(* Logix 5000 project; controller Project_Template vendor 1 type 14 code 106 rev 33.11; software revision 33.00 *)

TASK MainTask (continuous, watchdog 500 ms) : MainProgram

MODULES
   Local : vendor 1 type 14 code 106 (Compact 0, rev 33.11)
      Discrete_In_Slot_3 : 1769-IQ16 (Compact 3, rev 1.1, Input RPI 20 ms)
      Discrete_In_Slot_2 : 1769-IQ16 (Compact 2, rev 1.1, Input RPI 20 ms)
      Discrete_Out_Slot_5 : 1769-OW16 (Compact 5, rev 1.1, Output RPI 20 ms)
      Discrete_Out_Slot_4 : 1769-OW16 (Compact 4, rev 1.1, Output RPI 20 ms)
      ASCII_Slot_1 : vendor 1 type 109 code 66 (Compact 1, rev 2.1, Output RPI 2 ms)
END_MODULES

TYPE BCR_Data :
STRUCT
   LEN : DINT;
   DATA : SINT[9];
END_STRUCT
END_TYPE

TYPE Color_Data :
STRUCT
   LEN : DINT;
   DATA : SINT[4];
END_STRUCT
END_TYPE

VAR_GLOBAL   (* controller tags *)
   I_Auto_Mode_Selector : ALIAS FOR Local:2:I.Data.2;
   I_Barcode_Stop_Raised : ALIAS FOR Local:3:I.Data.1;
   I_Box_Ejector_Extended : ALIAS FOR Local:2:I.Data.4;
   I_Exit_Proxy : ALIAS FOR Local:3:I.Data.7;
   I_Reject_Cyl_Lowered : ALIAS FOR Local:3:I.Data.2;
   I_Reset_PB : ALIAS FOR Local:2:I.Data.3;
   I_Start_PB : ALIAS FOR Local:2:I.Data.0;
   I_Stop_PB : ALIAS FOR Local:2:I.Data.1;
   I_Vacuum_Head_at_Conveyor : ALIAS FOR Local:3:I.Data.0;
   I_Vacuum_Head_at_Magazine : ALIAS FOR Local:2:I.Data.15;
   I_Vacuum_Head_Extended : ALIAS FOR Local:2:I.Data.14;
   I_Vacuum_Head_Lowered : ALIAS FOR Local:2:I.Data.10;
   I_Vacuum_Head_Raised : ALIAS FOR Local:2:I.Data.9;
   I_Vacuum_Head_Retracted : ALIAS FOR Local:2:I.Data.13;
   I_Vacuum_Head_Rotated_CCW : ALIAS FOR Local:2:I.Data.11;
   I_Vacuum_Head_Rotated_CW : ALIAS FOR Local:2:I.Data.12;
   I_Vacuum_Sensor_On : ALIAS FOR Local:3:I.Data.8;
   O_Amber_Tower_Ind : ALIAS FOR Local:5:O.Data.9;
   O_Barcode_Stop_Raise : ALIAS FOR Local:4:O.Data.14;
   O_Box_Eject : ALIAS FOR Local:4:O.Data.0;
   O_Conveyor_On : ALIAS FOR Local:5:O.Data.5;
   O_Green_Tower_Ind : ALIAS FOR Local:5:O.Data.8;
   O_Red_Tower_Ind : ALIAS FOR Local:5:O.Data.10;
   O_Reject_Cyl_Extend : ALIAS FOR Local:5:O.Data.0;
   O_Reject_Cyl_Lower : ALIAS FOR Local:4:O.Data.15;
   O_Vacuum_Head_Extend : ALIAS FOR Local:4:O.Data.8;
   O_Vacuum_Head_Lower : ALIAS FOR Local:4:O.Data.5;
   O_Vacuum_Head_Rotate_CCW : ALIAS FOR Local:4:O.Data.7;
   O_Vacuum_Head_Rotate_CW : ALIAS FOR Local:4:O.Data.6;
   O_Vacuum_Head_to_Conveyor : ALIAS FOR Local:4:O.Data.9;
   O_Vacuum_Head_to_Magazine : ALIAS FOR Local:4:O.Data.10;
   O_Vacuum_Off : ALIAS FOR Local:5:O.Data.2;
   O_Vacuum_On : ALIAS FOR Local:5:O.Data.1;
END_VAR

PROGRAM MainProgram   (* main routine MainRoutine *)
VAR
   BCR_Good_Read : BOOL;
   BCR_Value : BCR_Data := '33320359$0D';
   Box_Filtered : BOOL;
   Color_Code : DINT := 2;
   Color_Value : Color_Data := '2';
   Delay_Timer : TIMER := (PRE := 3000);
   Fast_Flash_Off : TIMER := (PRE := 250, ACC := 182, EN := 1, TT := 1);
   Fast_Flash_On : TIMER := (PRE := 250, ACC := 250, EN := 1, DN := 1);
   Fast_Flasher : BOOL := 1;
   Filter_Done : BOOL := 1;
   Home_Verify : BOOL;
   Machine_Home : BOOL;
   New_Rx_ID : SINT := 26;
   Normal_Flash_Off : TIMER := (PRE := 500);
   Normal_Flash_On : TIMER := (PRE := 500, ACC := 432, EN := 1, TT := 1);
   Old_Rx_ID : SINT := 26;
   Prod_Cycl_Cntr : COUNTER := (ACC := 4, CU := 1, DN := 1);
   Prod_Cycl_end : BOOL := 1;
   Prod_Running : BOOL;
   Prod_Step : DINT;
   Prod_Test_Bit : DINT := -1;
   Production : BOOL;
   Regular_flasher : BOOL;
   Reject_Box : BOOL;
   Reset_Delay_Timer : TIMER[10] := ([0].PRE := 1000, [1].PRE := 1000, [2].PRE := 1000, [3].PRE := 1000, [4].PRE := 1000, [4].ACC := 1000, [4].EN := 1, [4].DN := 1, [5].PRE := 1000, [5].ACC := 1000, [5].EN := 1, [5].DN := 1);
   Reset_step : DINT;
   Reset_Test_Bit : DINT := -1;
   Resetting : BOOL;
   Rotate_timer : TIMER := (PRE := 500);
   Slow_Flash_Off : TIMER := (PRE := 1000);
   Slow_Flash_ON : TIMER := (PRE := 1000, ACC := 432, EN := 1, TT := 1);
   Slow_Flasher : BOOL;
   Stop_Bit : BOOL;
   Test_Bit : DINT;
END_VAR

ROUTINE a_Reset_Routine   (* ladder *)
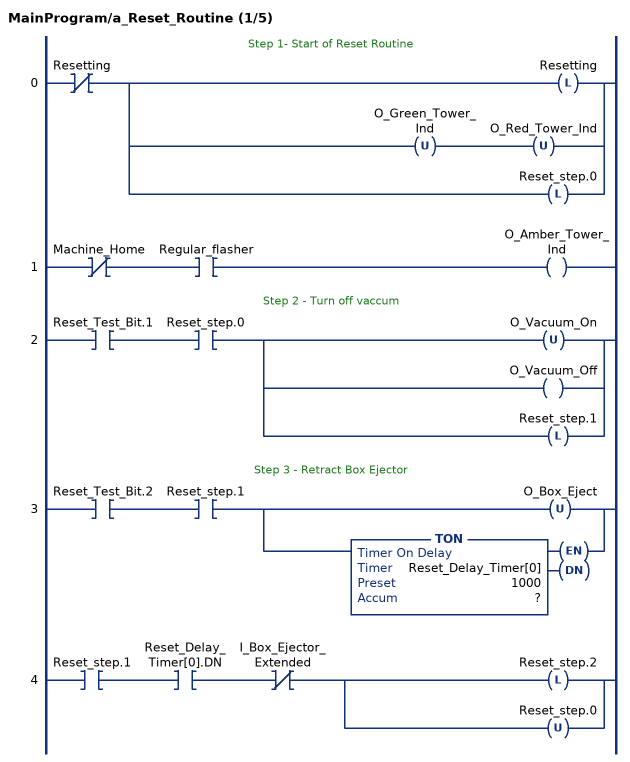
   // Step 1- Start of Reset Routine
   0: XIO(Resetting)[OTL(Resetting) ,OTU(O_Green_Tower_Ind) OTU(O_Red_Tower_Ind) ,OTL(Reset_step.0) ];
   1: XIO(Machine_Home)XIC(Regular_flasher)OTE(O_Amber_Tower_Ind);
   // Step 2 - Turn off vaccum
   2: XIC(Reset_Test_Bit.1)XIC(Reset_step.0)[OTU(O_Vacuum_On) ,OTE(O_Vacuum_Off) ,OTL(Reset_step.1) ];
   // Step 3 - Retract Box Ejector
   3: XIC(Reset_Test_Bit.2)XIC(Reset_step.1)[OTU(O_Box_Eject) ,TON(Reset_Delay_Timer[0],?,?) ];
   4: XIC(Reset_step.1)XIC(Reset_Delay_Timer[0].DN)XIO(I_Box_Ejector_Extended)[OTL(Reset_step.2) ,OTU(Reset_step.0) ];
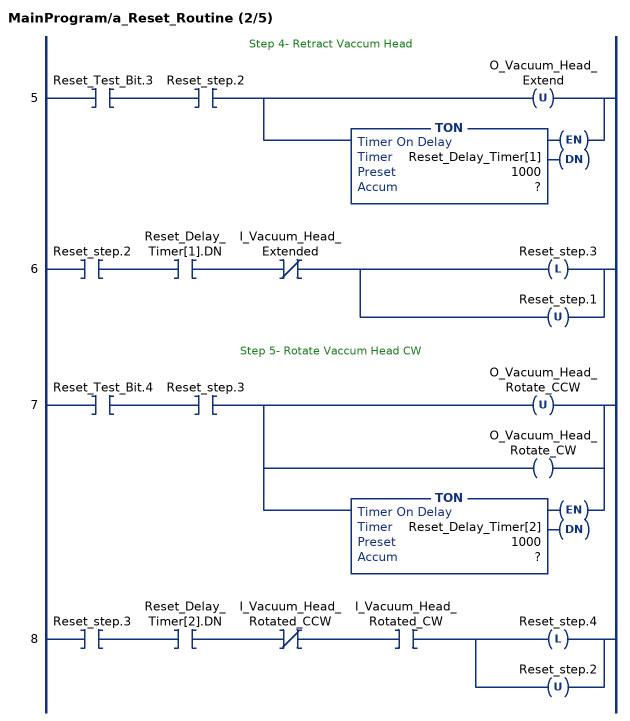
   // Step 4- Retract Vaccum Head
   5: XIC(Reset_Test_Bit.3)XIC(Reset_step.2)[OTU(O_Vacuum_Head_Extend) ,TON(Reset_Delay_Timer[1],?,?) ];
   6: XIC(Reset_step.2)XIC(Reset_Delay_Timer[1].DN)XIO(I_Vacuum_Head_Extended)[OTL(Reset_step.3) ,OTU(Reset_step.1) ];
   // Step 5- Rotate Vaccum Head CW
   7: XIC(Reset_Test_Bit.4)XIC(Reset_step.3)[OTU(O_Vacuum_Head_Rotate_CCW) ,OTE(O_Vacuum_Head_Rotate_CW) ,TON(Reset_Delay_Timer[2],?,?) ];
   8: XIC(Reset_step.3)XIC(Reset_Delay_Timer[2].DN)XIO(I_Vacuum_Head_Rotated_CCW)XIC(I_Vacuum_Head_Rotated_CW)[OTL(Reset_step.4) ,OTU(Reset_step.2) ];
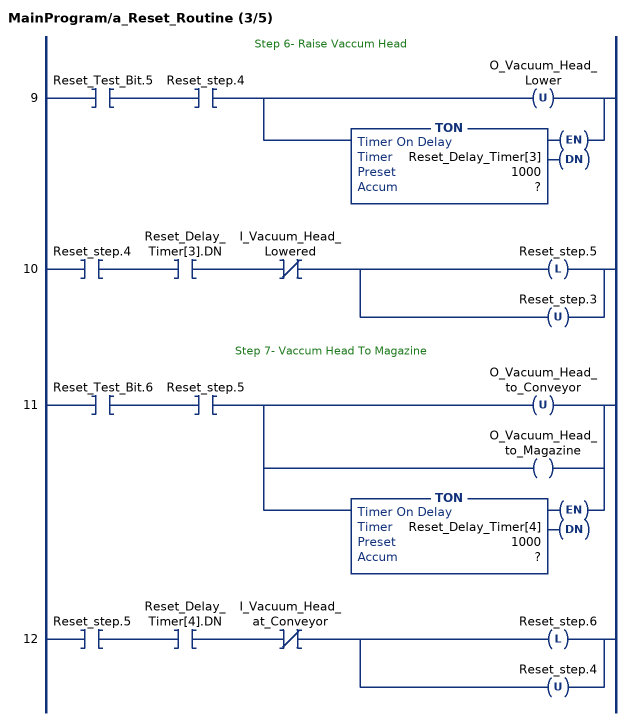
   // Step 6- Raise Vaccum Head
   9: XIC(Reset_Test_Bit.5)XIC(Reset_step.4)[OTU(O_Vacuum_Head_Lower) ,TON(Reset_Delay_Timer[3],?,?) ];
   10: XIC(Reset_step.4)XIC(Reset_Delay_Timer[3].DN)XIO(I_Vacuum_Head_Lowered)[OTL(Reset_step.5) ,OTU(Reset_step.3) ];
   // Step 7- Vaccum Head To Magazine
   11: XIC(Reset_Test_Bit.6)XIC(Reset_step.5)[OTU(O_Vacuum_Head_to_Conveyor) ,OTE(O_Vacuum_Head_to_Magazine) ,TON(Reset_Delay_Timer[4],?,?) ];
   12: XIC(Reset_step.5)XIC(Reset_Delay_Timer[4].DN)XIO(I_Vacuum_Head_at_Conveyor)[OTL(Reset_step.6) ,OTU(Reset_step.4) ];
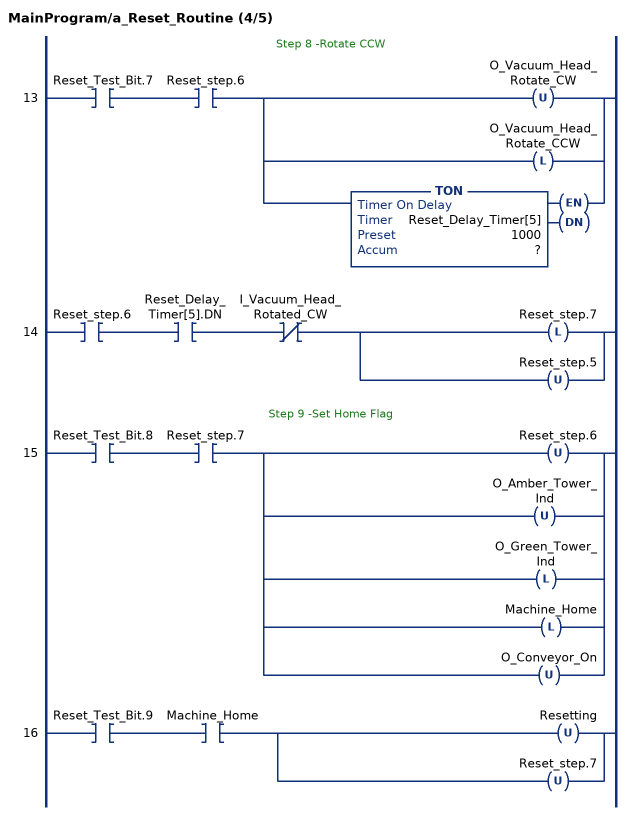
   // Step 8 -Rotate CCW
   13: XIC(Reset_Test_Bit.7)XIC(Reset_step.6)[OTU(O_Vacuum_Head_Rotate_CW) ,OTL(O_Vacuum_Head_Rotate_CCW) ,TON(Reset_Delay_Timer[5],?,?) ];
   14: XIC(Reset_step.6)XIC(Reset_Delay_Timer[5].DN)XIO(I_Vacuum_Head_Rotated_CW)[OTL(Reset_step.7) ,OTU(Reset_step.5) ];
   // Step 9 -Set Home Flag
   15: XIC(Reset_Test_Bit.8)XIC(Reset_step.7)[OTU(Reset_step.6) ,OTU(O_Amber_Tower_Ind) ,OTL(O_Green_Tower_Ind) ,OTL(Machine_Home) ,OTU(O_Conveyor_On) ];
   16: XIC(Reset_Test_Bit.9)XIC(Machine_Home)[OTU(Resetting) ,OTU(Reset_step.7) ];
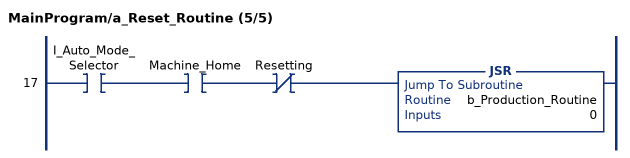
   17: XIC(I_Auto_Mode_Selector)XIC(Machine_Home)XIO(Resetting)JSR(b_Production_Routine,0);
END_ROUTINE

ROUTINE b_Production_Routine   (* ladder *)
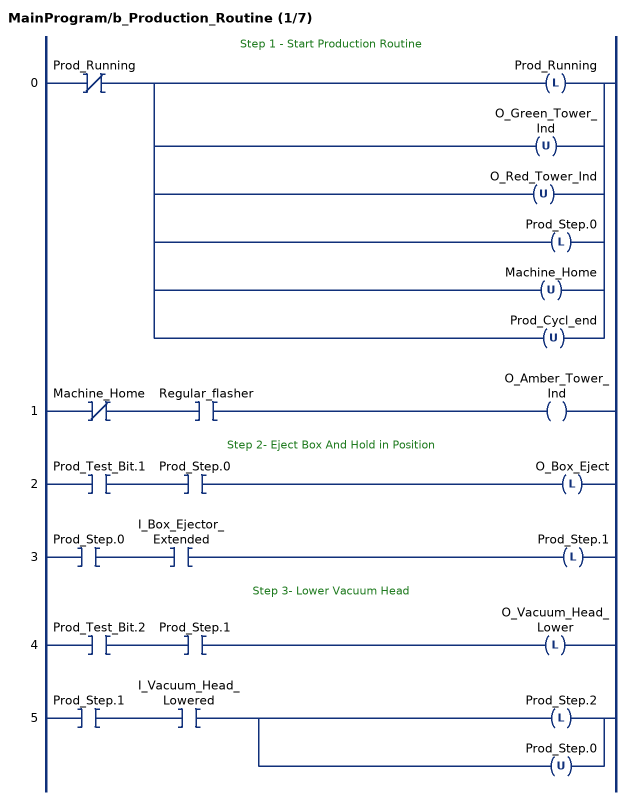
   // Step 1 - Start Production Routine
   0: XIO(Prod_Running)[OTL(Prod_Running) ,OTU(O_Green_Tower_Ind) ,OTU(O_Red_Tower_Ind) ,OTL(Prod_Step.0) ,OTU(Machine_Home) ,OTU(Prod_Cycl_end) ];
   1: XIO(Machine_Home)XIC(Regular_flasher)OTE(O_Amber_Tower_Ind);
   // Step 2- Eject Box And Hold in Position
   2: XIC(Prod_Test_Bit.1)XIC(Prod_Step.0)OTL(O_Box_Eject);
   3: XIC(Prod_Step.0)XIC(I_Box_Ejector_Extended)OTL(Prod_Step.1);
   // Step 3- Lower Vacuum Head
   4: XIC(Prod_Test_Bit.2)XIC(Prod_Step.1)OTL(O_Vacuum_Head_Lower);
   5: XIC(Prod_Step.1)XIC(I_Vacuum_Head_Lowered)[OTL(Prod_Step.2) ,OTU(Prod_Step.0) ];
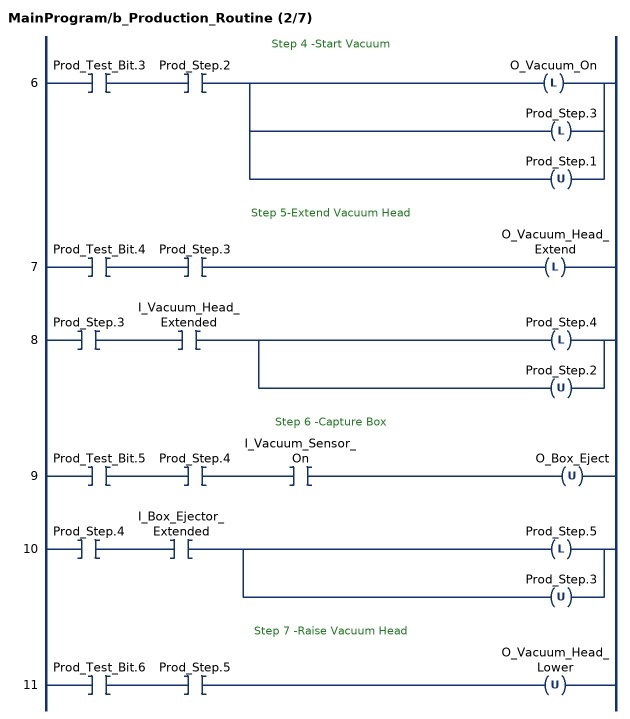
   // Step 4 -Start Vacuum
   6: XIC(Prod_Test_Bit.3)XIC(Prod_Step.2)[OTL(O_Vacuum_On) ,OTL(Prod_Step.3) ,OTU(Prod_Step.1) ];
   // Step 5-Extend Vacuum Head
   7: XIC(Prod_Test_Bit.4)XIC(Prod_Step.3)OTL(O_Vacuum_Head_Extend);
   8: XIC(Prod_Step.3)XIC(I_Vacuum_Head_Extended)[OTL(Prod_Step.4) ,OTU(Prod_Step.2) ];
   // Step 6 -Capture Box
   9: XIC(Prod_Test_Bit.5)XIC(Prod_Step.4)XIC(I_Vacuum_Sensor_On)OTU(O_Box_Eject);
   10: XIC(Prod_Step.4)XIC(I_Box_Ejector_Extended)[OTL(Prod_Step.5) ,OTU(Prod_Step.3) ];
   // Step 7 -Raise Vacuum Head
   11: XIC(Prod_Test_Bit.6)XIC(Prod_Step.5)OTU(O_Vacuum_Head_Lower);
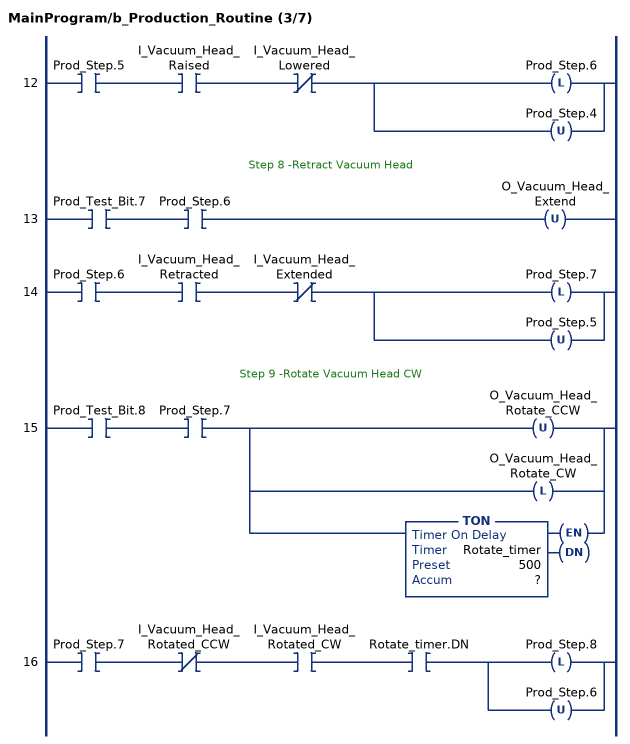
   12: XIC(Prod_Step.5)XIC(I_Vacuum_Head_Raised)XIO(I_Vacuum_Head_Lowered)[OTL(Prod_Step.6) ,OTU(Prod_Step.4) ];
   // Step 8 -Retract Vacuum Head
   13: XIC(Prod_Test_Bit.7)XIC(Prod_Step.6)OTU(O_Vacuum_Head_Extend);
   14: XIC(Prod_Step.6)XIC(I_Vacuum_Head_Retracted)XIO(I_Vacuum_Head_Extended)[OTL(Prod_Step.7) ,OTU(Prod_Step.5) ];
   // Step 9 -Rotate Vacuum Head CW
   15: XIC(Prod_Test_Bit.8)XIC(Prod_Step.7)[OTU(O_Vacuum_Head_Rotate_CCW) ,OTL(O_Vacuum_Head_Rotate_CW) ,TON(Rotate_timer,?,?) ];
   16: XIC(Prod_Step.7)XIO(I_Vacuum_Head_Rotated_CCW)XIC(I_Vacuum_Head_Rotated_CW)XIC(Rotate_timer.DN)[OTL(Prod_Step.8) ,OTU(Prod_Step.6) ];
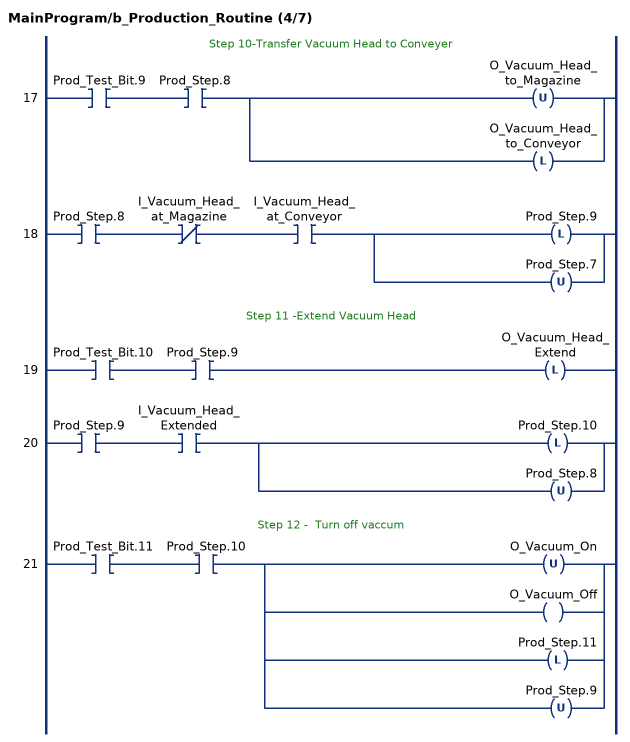
   // Step 10-Transfer Vacuum Head to Conveyer
   17: XIC(Prod_Test_Bit.9)XIC(Prod_Step.8)[OTU(O_Vacuum_Head_to_Magazine) ,OTL(O_Vacuum_Head_to_Conveyor) ];
   18: XIC(Prod_Step.8)XIO(I_Vacuum_Head_at_Magazine)XIC(I_Vacuum_Head_at_Conveyor)[OTL(Prod_Step.9) ,OTU(Prod_Step.7) ];
   // Step 11 -Extend Vacuum Head
   19: XIC(Prod_Test_Bit.10)XIC(Prod_Step.9)OTL(O_Vacuum_Head_Extend);
   20: XIC(Prod_Step.9)XIC(I_Vacuum_Head_Extended)[OTL(Prod_Step.10) ,OTU(Prod_Step.8) ];
   // Step 12 -  Turn off vaccum
   21: XIC(Prod_Test_Bit.11)XIC(Prod_Step.10)[OTU(O_Vacuum_On) ,OTE(O_Vacuum_Off) ,OTL(Prod_Step.11) ,OTU(Prod_Step.9) ];
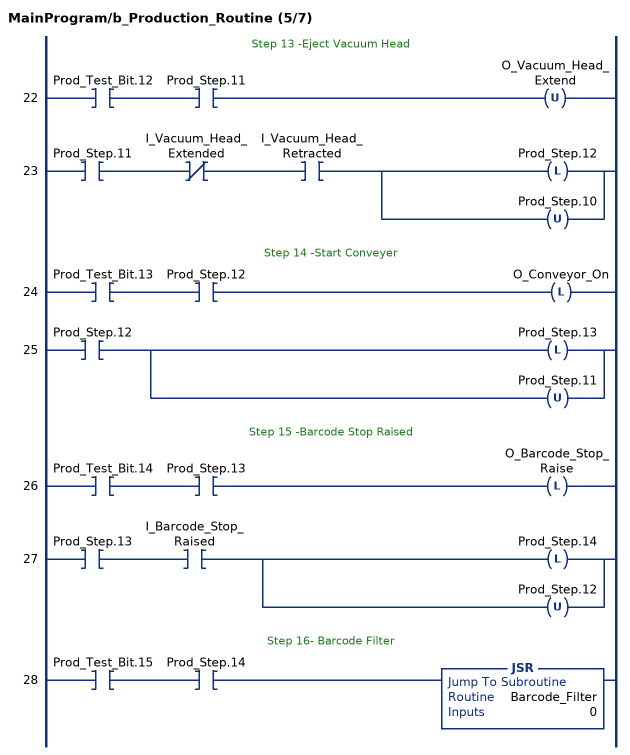
   // Step 13 -Eject Vacuum Head
   22: XIC(Prod_Test_Bit.12)XIC(Prod_Step.11)OTU(O_Vacuum_Head_Extend);
   23: XIC(Prod_Step.11)XIO(I_Vacuum_Head_Extended)XIC(I_Vacuum_Head_Retracted)[OTL(Prod_Step.12) ,OTU(Prod_Step.10) ];
   // Step 14 -Start Conveyer
   24: XIC(Prod_Test_Bit.13)XIC(Prod_Step.12)OTL(O_Conveyor_On);
   25: XIC(Prod_Step.12)[OTL(Prod_Step.13) ,OTU(Prod_Step.11) ];
   // Step 15 -Barcode Stop Raised
   26: XIC(Prod_Test_Bit.14)XIC(Prod_Step.13)OTL(O_Barcode_Stop_Raise);
   27: XIC(Prod_Step.13)XIC(I_Barcode_Stop_Raised)[OTL(Prod_Step.14) ,OTU(Prod_Step.12) ];
   // Step 16- Barcode Filter
   28: XIC(Prod_Test_Bit.15)XIC(Prod_Step.14)JSR(Barcode_Filter,0);
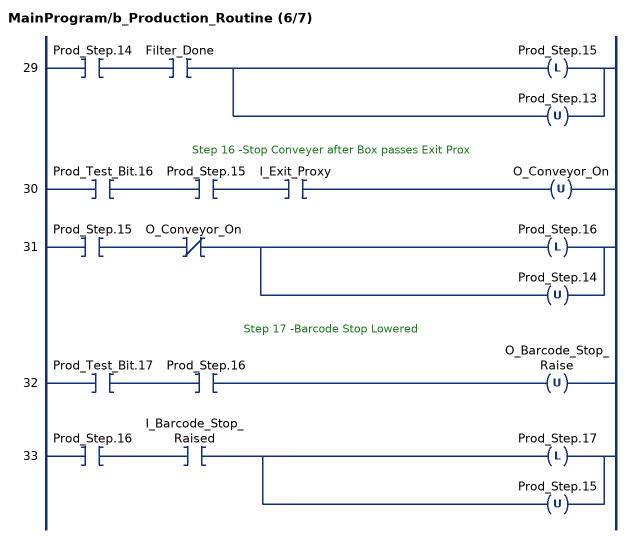
   29: XIC(Prod_Step.14)XIC(Filter_Done)[OTL(Prod_Step.15) ,OTU(Prod_Step.13) ];
   // Step 16 -Stop Conveyer after Box passes Exit Prox
   30: XIC(Prod_Test_Bit.16)XIC(Prod_Step.15)XIC(I_Exit_Proxy)OTU(O_Conveyor_On);
   31: XIC(Prod_Step.15)XIO(O_Conveyor_On)[OTL(Prod_Step.16) ,OTU(Prod_Step.14) ];
   // Step 17 -Barcode Stop Lowered
   32: XIC(Prod_Test_Bit.17)XIC(Prod_Step.16)OTU(O_Barcode_Stop_Raise);
   33: XIC(Prod_Step.16)XIC(I_Barcode_Stop_Raised)[OTL(Prod_Step.17) ,OTU(Prod_Step.15) ];
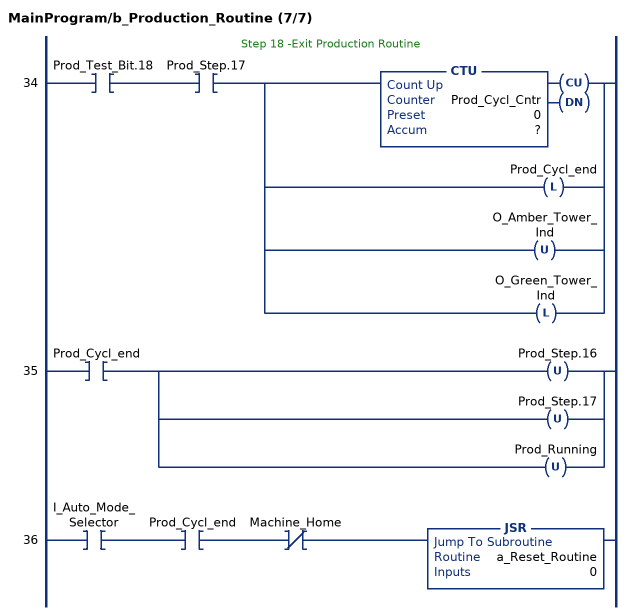
   // Step 18 -Exit Production Routine
   34: XIC(Prod_Test_Bit.18)XIC(Prod_Step.17)[CTU(Prod_Cycl_Cntr,?,?) ,OTL(Prod_Cycl_end) ,OTU(O_Amber_Tower_Ind) ,OTL(O_Green_Tower_Ind) ];
   35: XIC(Prod_Cycl_end)[OTU(Prod_Step.16) ,OTU(Prod_Step.17) ,OTU(Prod_Running) ];
   36: XIC(I_Auto_Mode_Selector)XIC(Prod_Cycl_end)XIO(Machine_Home)JSR(a_Reset_Routine,0);
END_ROUTINE

ROUTINE Barcode_Filter   (* ladder *)
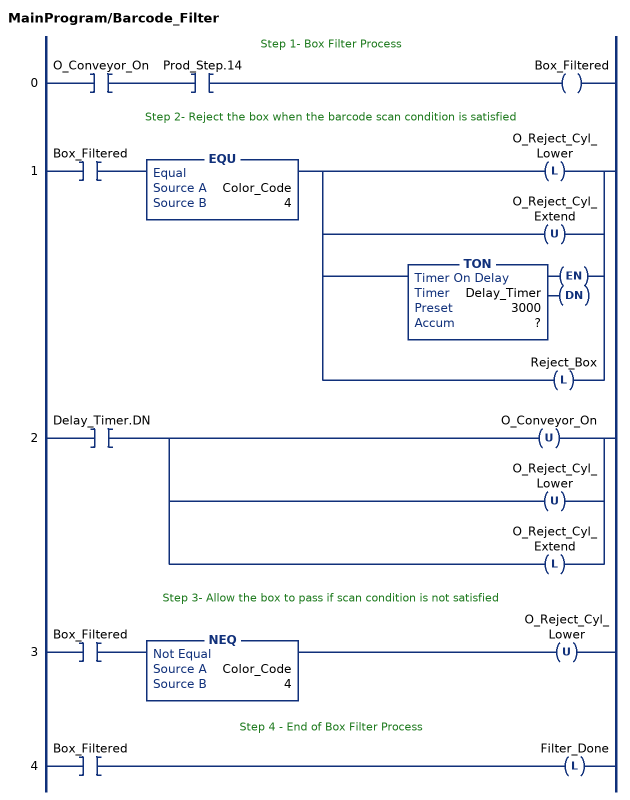
   // Step 1- Box Filter Process
   0: XIC(O_Conveyor_On)XIC(Prod_Step.14)OTE(Box_Filtered);
   // Step 2- Reject the box when the barcode scan condition is satisfied
   1: XIC(Box_Filtered)EQU(Color_Code,4)[OTL(O_Reject_Cyl_Lower) ,OTU(O_Reject_Cyl_Extend) ,TON(Delay_Timer,?,?) ,OTL(Reject_Box) ];
   2: XIC(Delay_Timer.DN)[OTU(O_Conveyor_On) ,OTU(O_Reject_Cyl_Lower) ,OTL(O_Reject_Cyl_Extend) ];
   // Step 3- Allow the box to pass if scan condition is not satisfied
   3: XIC(Box_Filtered)NEQ(Color_Code,4)OTU(O_Reject_Cyl_Lower);
   // Step 4 - End of Box Filter Process
   4: XIC(Box_Filtered)OTL(Filter_Done);
END_ROUTINE

ROUTINE Barcode_Read   (* ladder *)
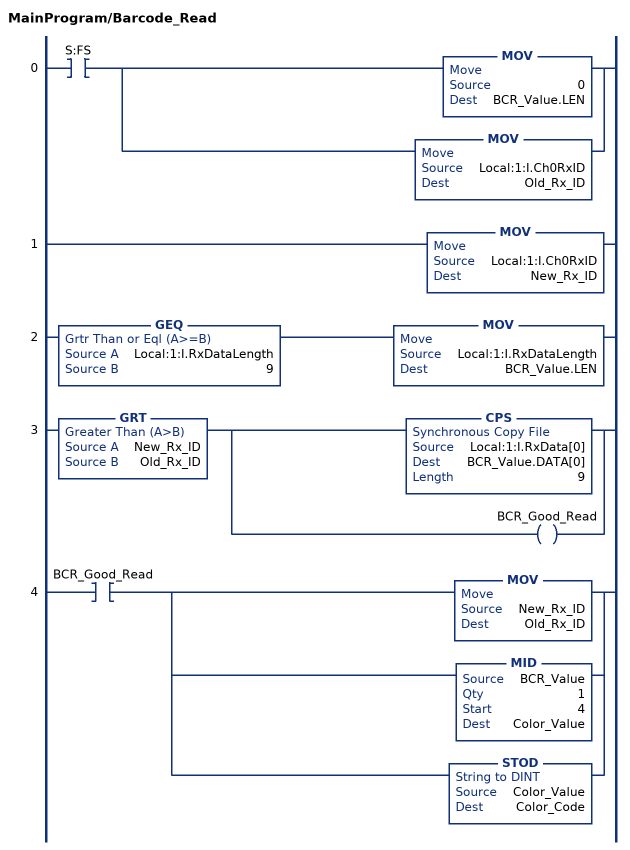
   0: XIC(S:FS)[MOV(0,BCR_Value.LEN) ,MOV(Local:1:I.Ch0RxID,Old_Rx_ID) ];
   1: MOV(Local:1:I.Ch0RxID,New_Rx_ID);
   2: GEQ(Local:1:I.RxDataLength,9)MOV(Local:1:I.RxDataLength,BCR_Value.LEN);
   3: GRT(New_Rx_ID,Old_Rx_ID)[CPS(Local:1:I.RxData[0],BCR_Value.DATA[0],9) ,OTE(BCR_Good_Read) ];
   4: XIC(BCR_Good_Read)[MOV(New_Rx_ID,Old_Rx_ID) ,MID(BCR_Value,1,4,Color_Value) ,STOD(Color_Value,Color_Code) ];
END_ROUTINE

ROUTINE Home_Verification   (* ladder *)
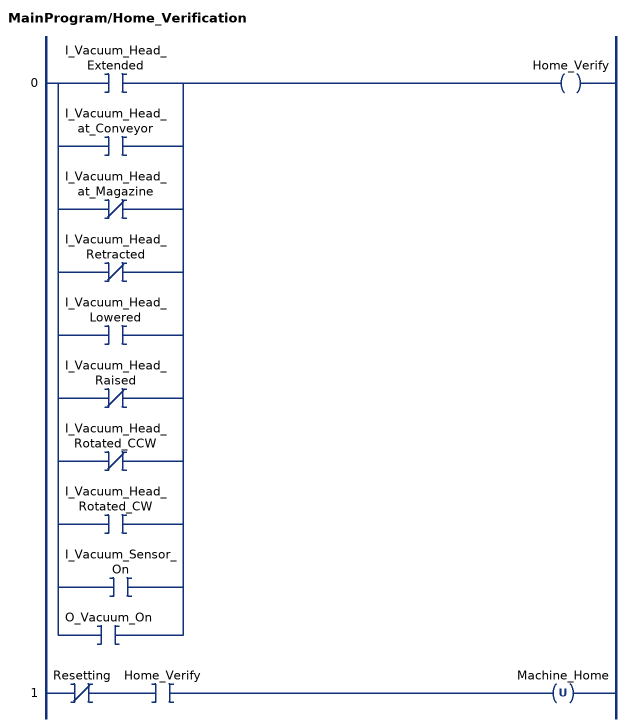
   0: [XIC(I_Vacuum_Head_Extended) ,XIC(I_Vacuum_Head_at_Conveyor) ,XIO(I_Vacuum_Head_at_Magazine) ,XIO(I_Vacuum_Head_Retracted) ,XIC(I_Vacuum_Head_Lowered) ,XIO(I_Vacuum_Head_Raised) ,XIO(I_Vacuum_Head_Rotated_CCW) ,XIC(I_Vacuum_Head_Rotated_CW) ,XIC(I_Vacuum_Sensor_On) ,XIC(O_Vacuum_On) ]OTE(Home_Verify);
   1: XIO(Resetting)XIC(Home_Verify)OTU(Machine_Home);
END_ROUTINE

ROUTINE MainRoutine   (* ladder *)
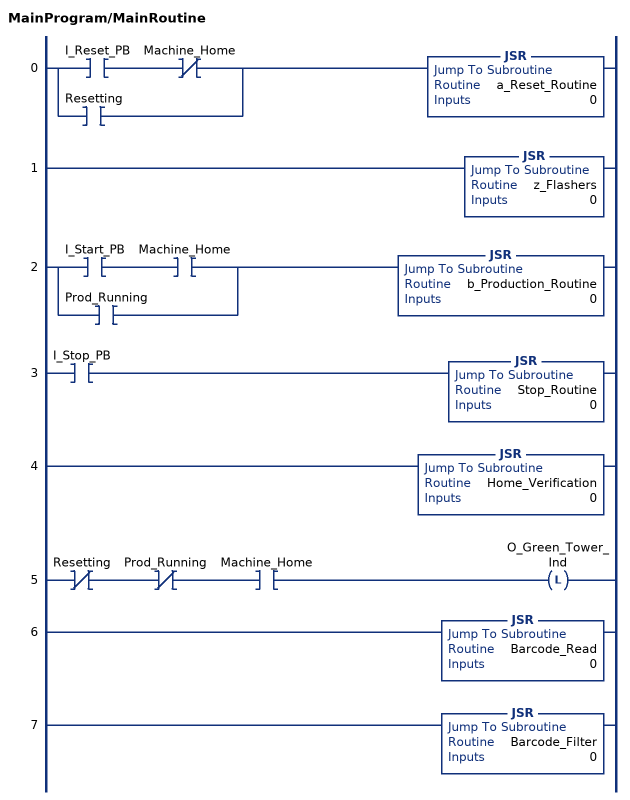
   0: [XIC(I_Reset_PB) XIO(Machine_Home) ,XIC(Resetting) ]JSR(a_Reset_Routine,0);
   1: JSR(z_Flashers,0);
   2: [XIC(I_Start_PB) XIC(Machine_Home) ,XIC(Prod_Running) ]JSR(b_Production_Routine,0);
   3: XIC(I_Stop_PB)JSR(Stop_Routine,0);
   4: JSR(Home_Verification,0);
   5: XIO(Resetting)XIO(Prod_Running)XIC(Machine_Home)OTL(O_Green_Tower_Ind);
   6: JSR(Barcode_Read,0);
   7: JSR(Barcode_Filter,0);
END_ROUTINE

ROUTINE Stop_Routine   (* ladder *)
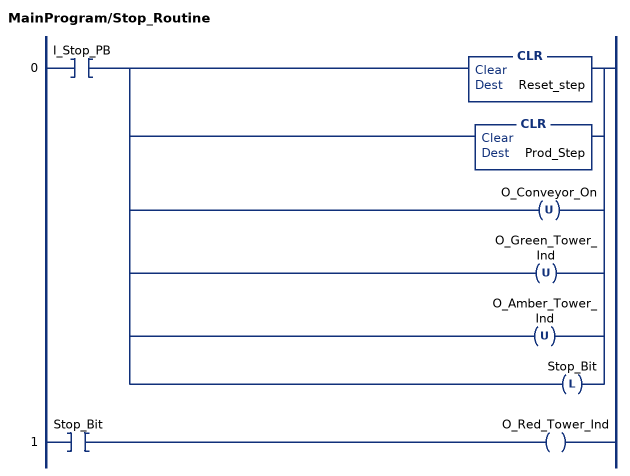
   0: XIC(I_Stop_PB)[CLR(Reset_step) ,CLR(Prod_Step) ,OTU(O_Conveyor_On) ,OTU(O_Green_Tower_Ind) ,OTU(O_Amber_Tower_Ind) ,OTL(Stop_Bit) ];
   1: XIC(Stop_Bit)OTE(O_Red_Tower_Ind);
END_ROUTINE

ROUTINE z_Flashers   (* ladder *)
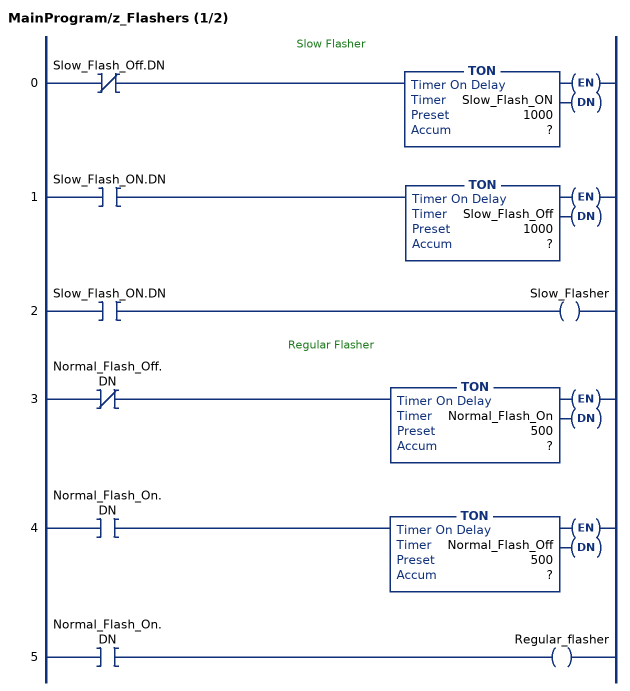
   // Slow Flasher
   0: XIO(Slow_Flash_Off.DN)TON(Slow_Flash_ON,?,?);
   1: XIC(Slow_Flash_ON.DN)TON(Slow_Flash_Off,?,?);
   2: XIC(Slow_Flash_ON.DN)OTE(Slow_Flasher);
   // Regular Flasher
   3: XIO(Normal_Flash_Off.DN)TON(Normal_Flash_On,?,?);
   4: XIC(Normal_Flash_On.DN)TON(Normal_Flash_Off,?,?);
   5: XIC(Normal_Flash_On.DN)OTE(Regular_flasher);
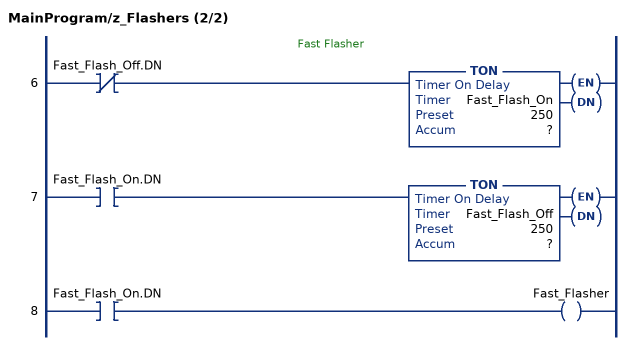
   // Fast Flasher
   6: XIO(Fast_Flash_Off.DN)TON(Fast_Flash_On,?,?);
   7: XIC(Fast_Flash_On.DN)TON(Fast_Flash_Off,?,?);
   8: XIC(Fast_Flash_On.DN)OTE(Fast_Flasher);
END_ROUTINE
END_PROGRAM
